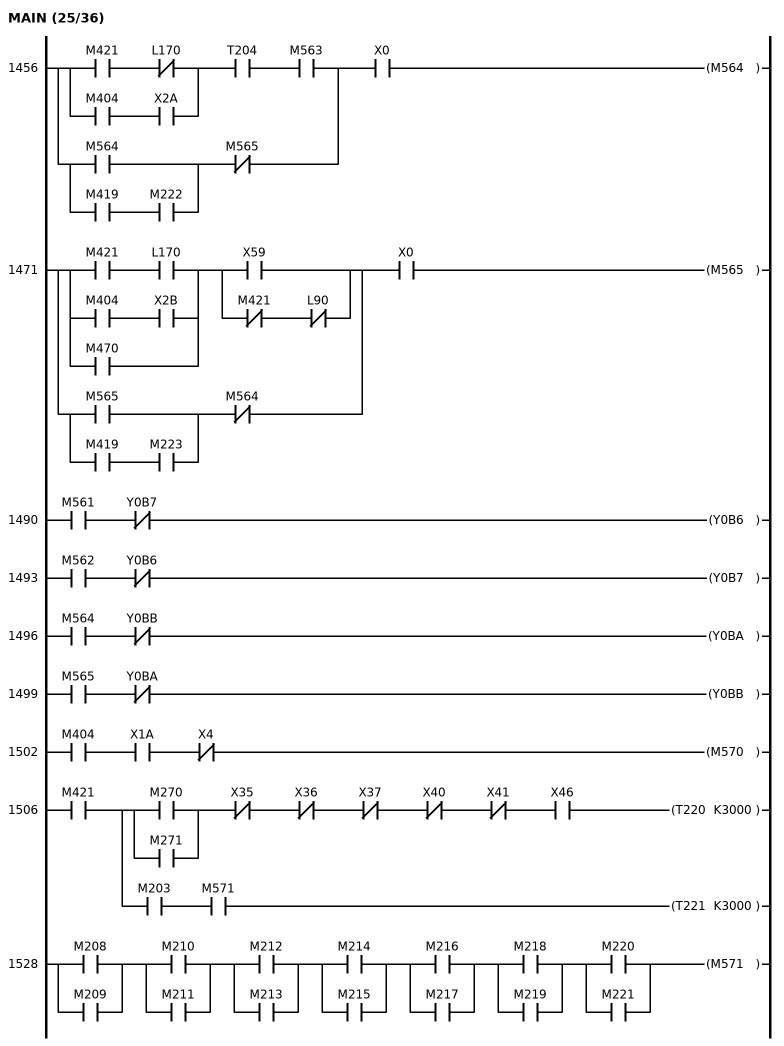
[picture p24: ladder of MAIN, rungs at steps 1456 to 1528]
1456  LD      M421
      ANI     L170
      LD      M404
      AND     X2A
      ORB
      AND     T204
      AND     M563
      LD      M564
      LD      M419
      AND     M222
      ORB
      ANI     M565
      ORB
      AND     X0
      OUT     M564
1471  LD      M421
      AND     L170
      LD      M404
      AND     X2B
      ORB
      OR      M470
      LD      X59
      LDI     M421
      ANI     L90
      ORB
      ANB
      LD      M565
      LD      M419
      AND     M223
      ORB
      ANI     M564
      ORB
      AND     X0
      OUT     M565
1490  LD      M561
      ANI     Y0B7
      OUT     Y0B6
1493  LD      M562
      ANI     Y0B6
      OUT     Y0B7
1496  LD      M564
      ANI     Y0BB
      OUT     Y0BA
1499  LD      M565
      ANI     Y0BA
      OUT     Y0BB
1502  LD      M404
      AND     X1A
      ANI     X4
      OUT     M570
1506  LD      M421
      MPS
      LD      M270
      OR      M271
      ANB
      ANI     X35
      ANI     X36
      ANI     X37
      ANI     X40
      ANI     X41
      AND     X46
      OUT     T220 K3000
      MPP
      AND     M203
      AND     M571
      OUT     T221 K3000
1528  LD      M208
      OR      M209
      LD      M210
      OR      M211
      ANB
      LD      M212
      OR      M213
      ANB
      LD      M214
      OR      M215
      ANB
      LD      M216
      OR      M217
      ANB
      LD      M218
      OR      M219
      ANB
      LD      M220
      OR      M221
      ANB
      OUT     M571
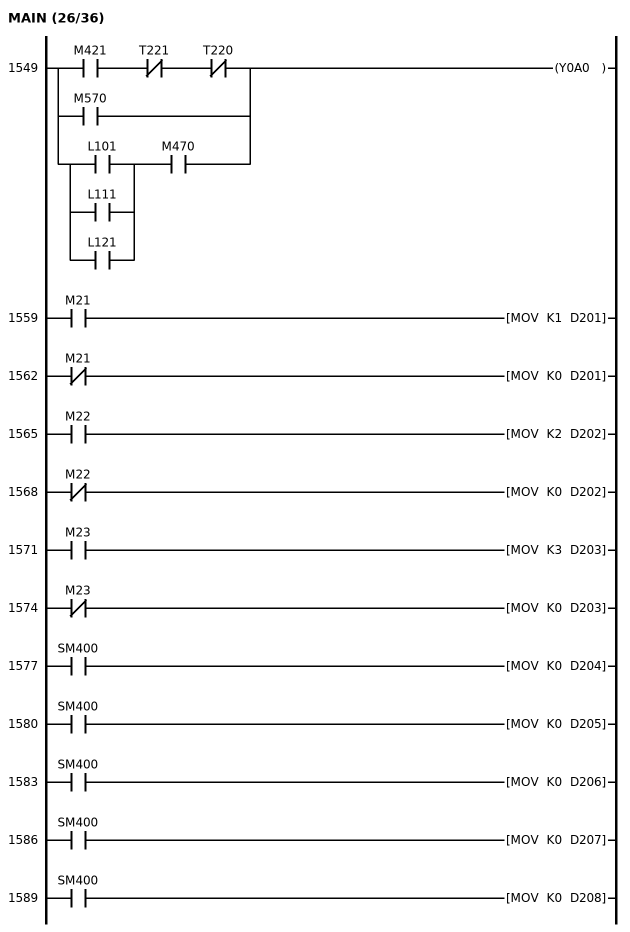
1549  LD      M421
      ANI     T221
      ANI     T220
      OR      M570
      LD      L101
      OR      L111
      OR      L121
      AND     M470
      ORB
      OUT     Y0A0
1559  LD      M21
      MOV     K1 D201
1562  LDI     M21
      MOV     K0 D201
1565  LD      M22
      MOV     K2 D202
1568  LDI     M22
      MOV     K0 D202
1571  LD      M23
      MOV     K3 D203
1574  LDI     M23
      MOV     K0 D203
1577  LD      SM400
      MOV     K0 D204
1580  LD      SM400
      MOV     K0 D205
1583  LD      SM400
      MOV     K0 D206
1586  LD      SM400
      MOV     K0 D207
1589  LD      SM400
      MOV     K0 D208
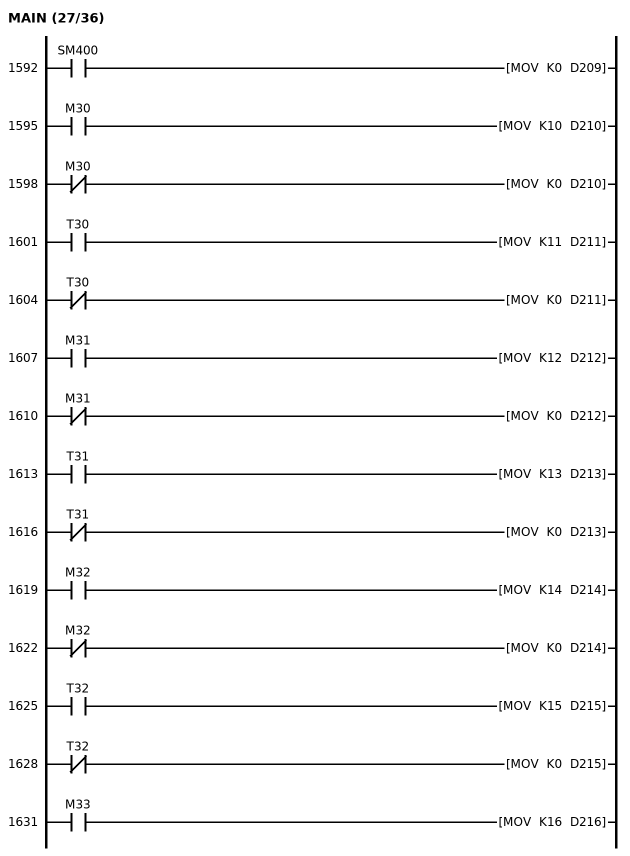
1592  LD      SM400
      MOV     K0 D209
1595  LD      M30
      MOV     K10 D210
1598  LDI     M30
      MOV     K0 D210
1601  LD      T30
      MOV     K11 D211
1604  LDI     T30
      MOV     K0 D211
1607  LD      M31
      MOV     K12 D212
1610  LDI     M31
      MOV     K0 D212
1613  LD      T31
      MOV     K13 D213
1616  LDI     T31
      MOV     K0 D213
1619  LD      M32
      MOV     K14 D214
1622  LDI     M32
      MOV     K0 D214
1625  LD      T32
      MOV     K15 D215
1628  LDI     T32
      MOV     K0 D215
1631  LD      M33
      MOV     K16 D216
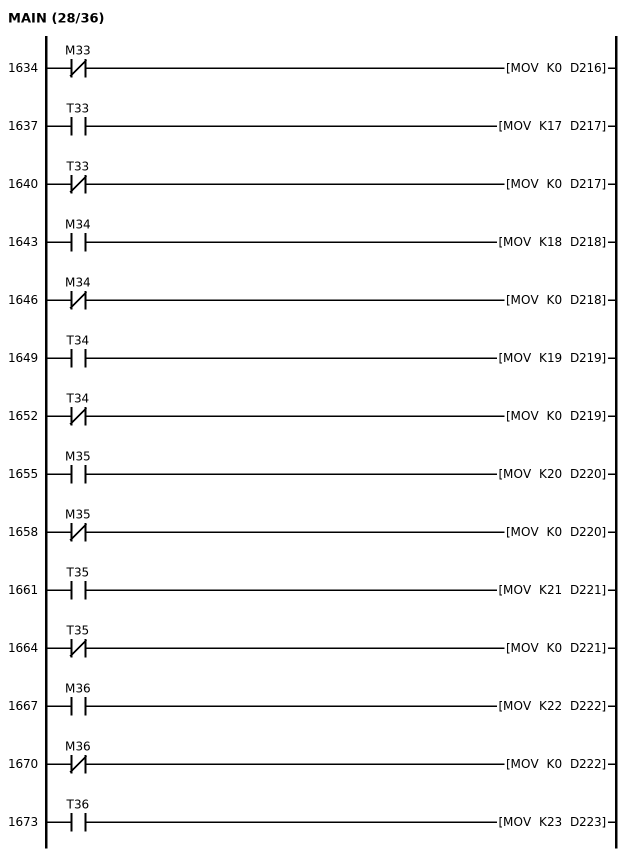
1634  LDI     M33
      MOV     K0 D216
1637  LD      T33
      MOV     K17 D217
1640  LDI     T33
      MOV     K0 D217
1643  LD      M34
      MOV     K18 D218
1646  LDI     M34
      MOV     K0 D218
1649  LD      T34
      MOV     K19 D219
1652  LDI     T34
      MOV     K0 D219
1655  LD      M35
      MOV     K20 D220
1658  LDI     M35
      MOV     K0 D220
1661  LD      T35
      MOV     K21 D221
1664  LDI     T35
      MOV     K0 D221
1667  LD      M36
      MOV     K22 D222
1670  LDI     M36
      MOV     K0 D222
1673  LD      T36
      MOV     K23 D223
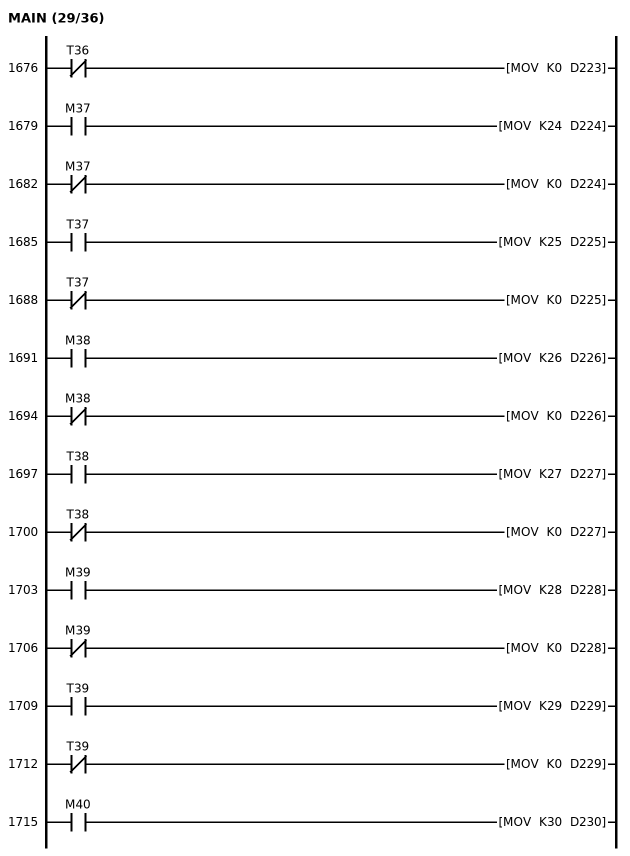
1676  LDI     T36
      MOV     K0 D223
1679  LD      M37
      MOV     K24 D224
1682  LDI     M37
      MOV     K0 D224
1685  LD      T37
      MOV     K25 D225
1688  LDI     T37
      MOV     K0 D225
1691  LD      M38
      MOV     K26 D226
1694  LDI     M38
      MOV     K0 D226
1697  LD      T38
      MOV     K27 D227
1700  LDI     T38
      MOV     K0 D227
1703  LD      M39
      MOV     K28 D228
1706  LDI     M39
      MOV     K0 D228
1709  LD      T39
      MOV     K29 D229
1712  LDI     T39
      MOV     K0 D229
1715  LD      M40
      MOV     K30 D230
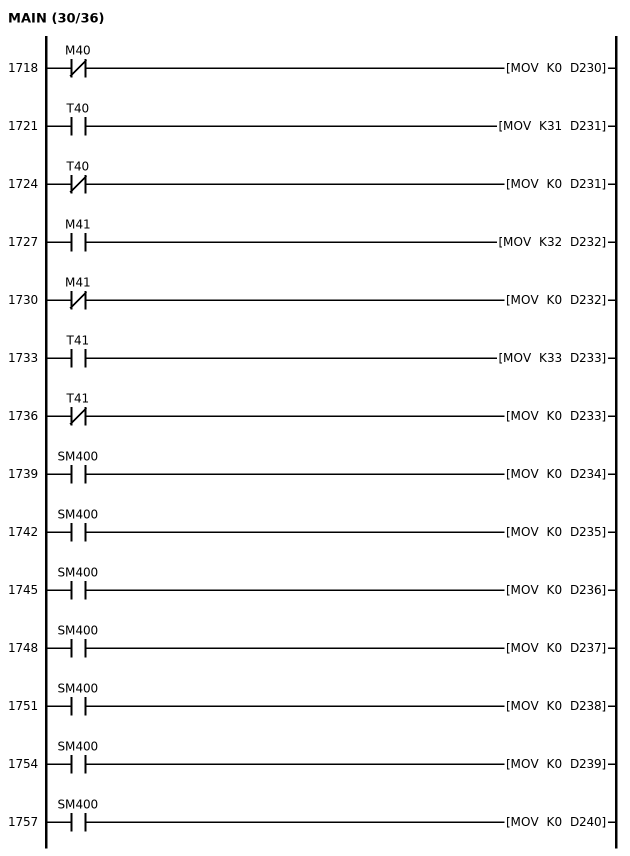
1718  LDI     M40
      MOV     K0 D230
1721  LD      T40
      MOV     K31 D231
1724  LDI     T40
      MOV     K0 D231
1727  LD      M41
      MOV     K32 D232
1730  LDI     M41
      MOV     K0 D232
1733  LD      T41
      MOV     K33 D233
1736  LDI     T41
      MOV     K0 D233
1739  LD      SM400
      MOV     K0 D234
1742  LD      SM400
      MOV     K0 D235
1745  LD      SM400
      MOV     K0 D236
1748  LD      SM400
      MOV     K0 D237
1751  LD      SM400
      MOV     K0 D238
1754  LD      SM400
      MOV     K0 D239
1757  LD      SM400
      MOV     K0 D240
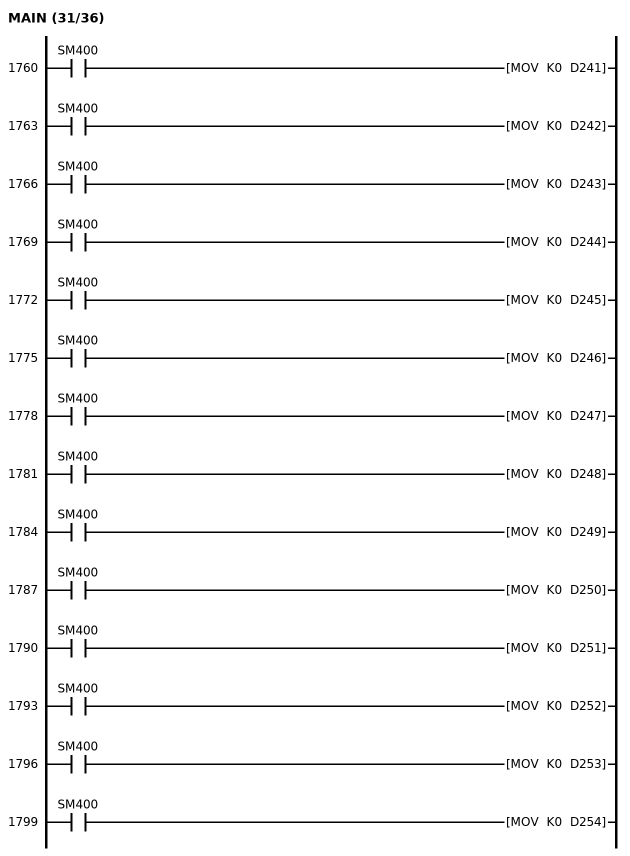
1760  LD      SM400
      MOV     K0 D241
1763  LD      SM400
      MOV     K0 D242
1766  LD      SM400
      MOV     K0 D243
1769  LD      SM400
      MOV     K0 D244
1772  LD      SM400
      MOV     K0 D245
1775  LD      SM400
      MOV     K0 D246
1778  LD      SM400
      MOV     K0 D247
1781  LD      SM400
      MOV     K0 D248
1784  LD      SM400
      MOV     K0 D249
1787  LD      SM400
      MOV     K0 D250
1790  LD      SM400
      MOV     K0 D251
1793  LD      SM400
      MOV     K0 D252
1796  LD      SM400
      MOV     K0 D253
1799  LD      SM400
      MOV     K0 D254
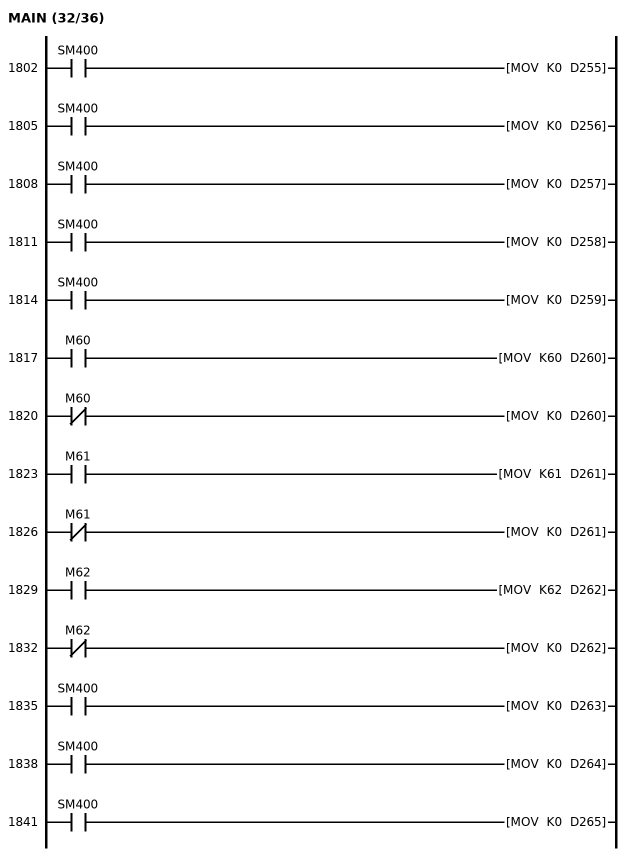
1802  LD      SM400
      MOV     K0 D255
1805  LD      SM400
      MOV     K0 D256
1808  LD      SM400
      MOV     K0 D257
1811  LD      SM400
      MOV     K0 D258
1814  LD      SM400
      MOV     K0 D259
1817  LD      M60
      MOV     K60 D260
1820  LDI     M60
      MOV     K0 D260
1823  LD      M61
      MOV     K61 D261
1826  LDI     M61
      MOV     K0 D261
1829  LD      M62
      MOV     K62 D262
1832  LDI     M62
      MOV     K0 D262
1835  LD      SM400
      MOV     K0 D263
1838  LD      SM400
      MOV     K0 D264
1841  LD      SM400
      MOV     K0 D265
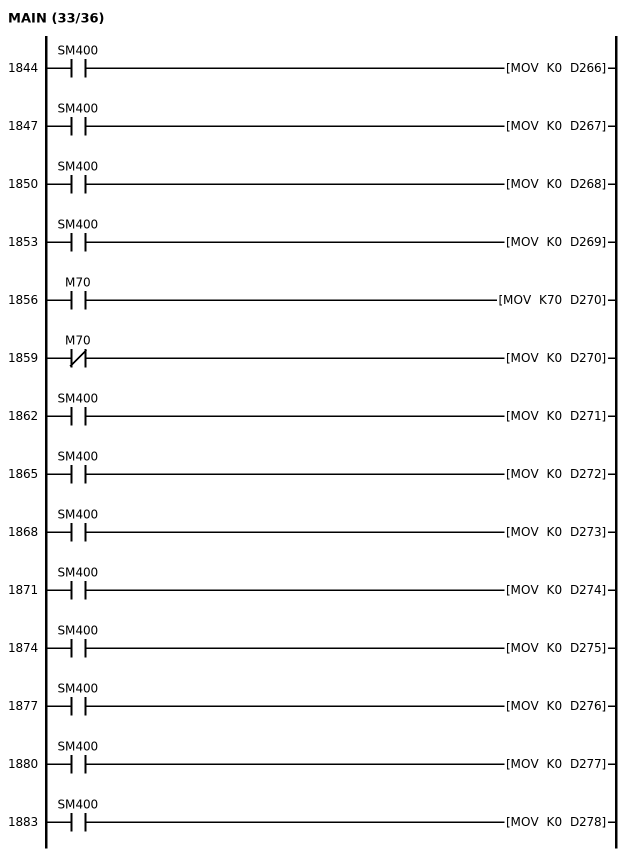
1844  LD      SM400
      MOV     K0 D266
1847  LD      SM400
      MOV     K0 D267
1850  LD      SM400
      MOV     K0 D268
1853  LD      SM400
      MOV     K0 D269
1856  LD      M70
      MOV     K70 D270
1859  LDI     M70
      MOV     K0 D270
1862  LD      SM400
      MOV     K0 D271
1865  LD      SM400
      MOV     K0 D272
1868  LD      SM400
      MOV     K0 D273
1871  LD      SM400
      MOV     K0 D274
1874  LD      SM400
      MOV     K0 D275
1877  LD      SM400
      MOV     K0 D276
1880  LD      SM400
      MOV     K0 D277
1883  LD      SM400
      MOV     K0 D278
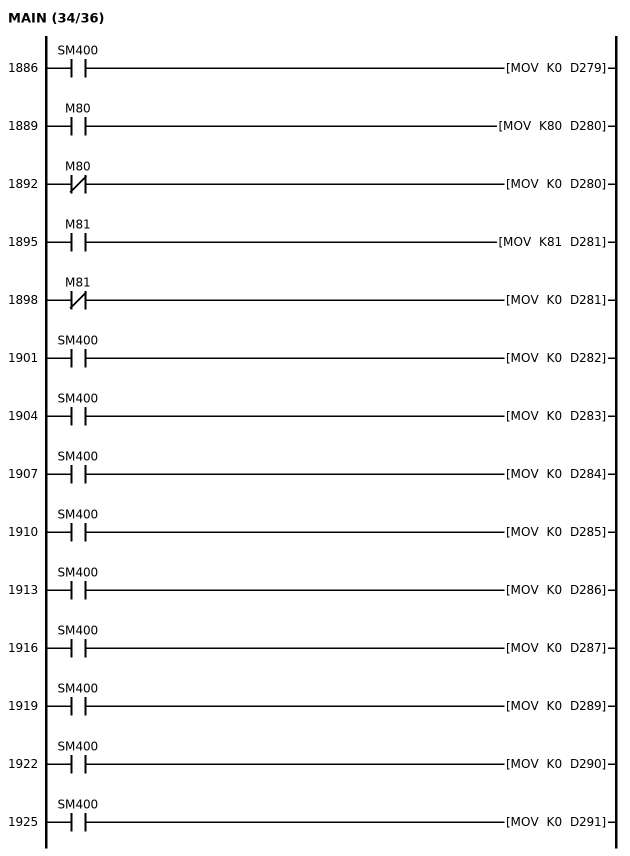
1886  LD      SM400
      MOV     K0 D279
1889  LD      M80
      MOV     K80 D280
1892  LDI     M80
      MOV     K0 D280
1895  LD      M81
      MOV     K81 D281
1898  LDI     M81
      MOV     K0 D281
1901  LD      SM400
      MOV     K0 D282
1904  LD      SM400
      MOV     K0 D283
1907  LD      SM400
      MOV     K0 D284
1910  LD      SM400
      MOV     K0 D285
1913  LD      SM400
      MOV     K0 D286
1916  LD      SM400
      MOV     K0 D287
1919  LD      SM400
      MOV     K0 D289
1922  LD      SM400
      MOV     K0 D290
1925  LD      SM400
      MOV     K0 D291
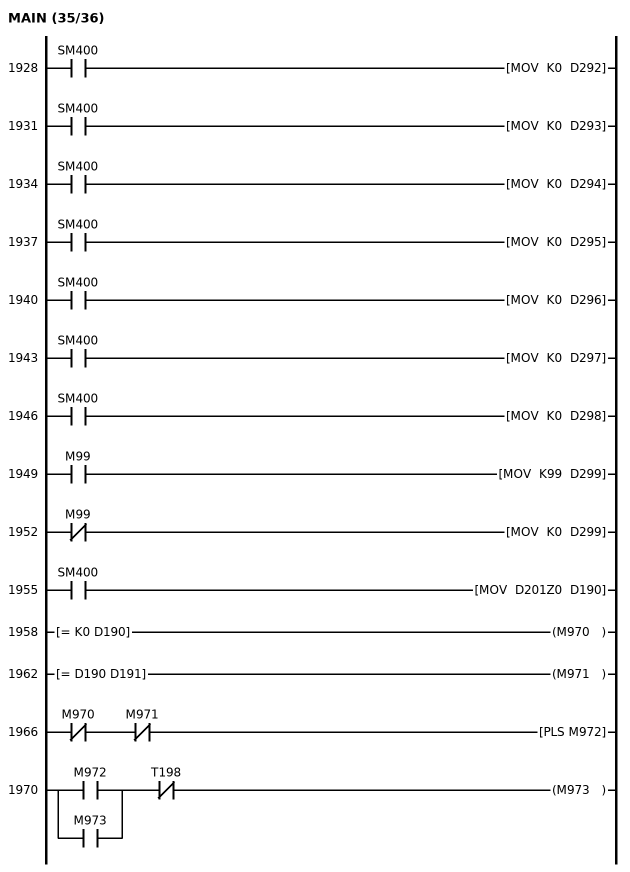
1928  LD      SM400
      MOV     K0 D292
1931  LD      SM400
      MOV     K0 D293
1934  LD      SM400
      MOV     K0 D294
1937  LD      SM400
      MOV     K0 D295
1940  LD      SM400
      MOV     K0 D296
1943  LD      SM400
      MOV     K0 D297
1946  LD      SM400
      MOV     K0 D298
1949  LD      M99
      MOV     K99 D299
1952  LDI     M99
      MOV     K0 D299
1955  LD      SM400
      MOV     D201Z0 D190
1958  LD=     K0 D190
      OUT     M970
1962  LD=     D190 D191
      OUT     M971
1966  LDI     M970
      ANI     M971
      PLS     M972
1970  LD      M972
      OR      M973
      ANI     T198
      OUT     M973
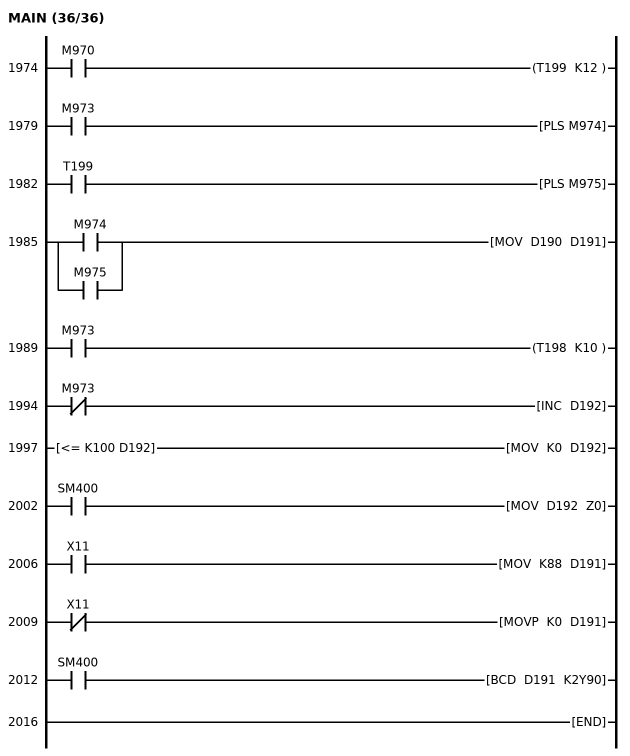
1974  LD      M970
      OUT     T199 K12
1979  LD      M973
      PLS     M974
1982  LD      T199
      PLS     M975
1985  LD      M974
      OR      M975
      MOV     D190 D191
1989  LD      M973
      OUT     T198 K10
1994  LDI     M973
      INC     D192
1997  LD<=    K100 D192
      MOV     K0 D192
2002  LD      SM400
      MOV     D192 Z0
2006  LD      X11
      MOV     K88 D191
2009  LDI     X11
      MOVP    K0 D191
2012  LD      SM400
      BCD     D191 K2Y90
2016  END
END_PROGRAM
